// Mitsubishi GX Works2 project: 램프4   PLC: Q02/Q02H

PROGRAM MAIN
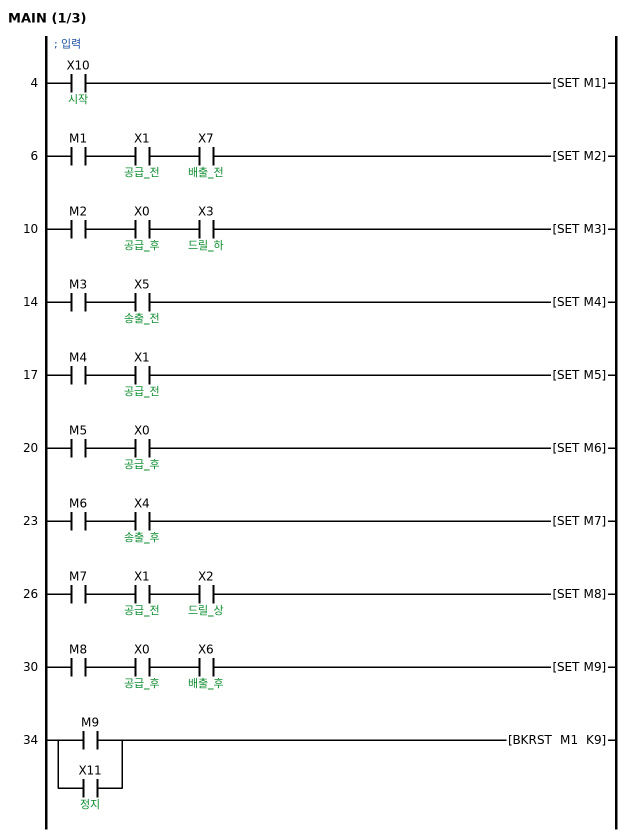
; 입력
4     LD      X10  ; 시작
      SET     M1
6     LD      M1
      AND     X1  ; 공급_전
      AND     X7  ; 배출_전
      SET     M2
10    LD      M2
      AND     X0  ; 공급_후
      AND     X3  ; 드릴_하
      SET     M3
14    LD      M3
      AND     X5  ; 송출_전
      SET     M4
17    LD      M4
      AND     X1  ; 공급_전
      SET     M5
20    LD      M5
      AND     X0  ; 공급_후
      SET     M6
23    LD      M6
      AND     X4  ; 송출_후
      SET     M7
26    LD      M7
      AND     X1  ; 공급_전
      AND     X2  ; 드릴_상
      SET     M8
30    LD      M8
      AND     X0  ; 공급_후
      AND     X6  ; 배출_후
      SET     M9
34    LD      M9
      OR      X11  ; 정지
      BKRST   M1 K9
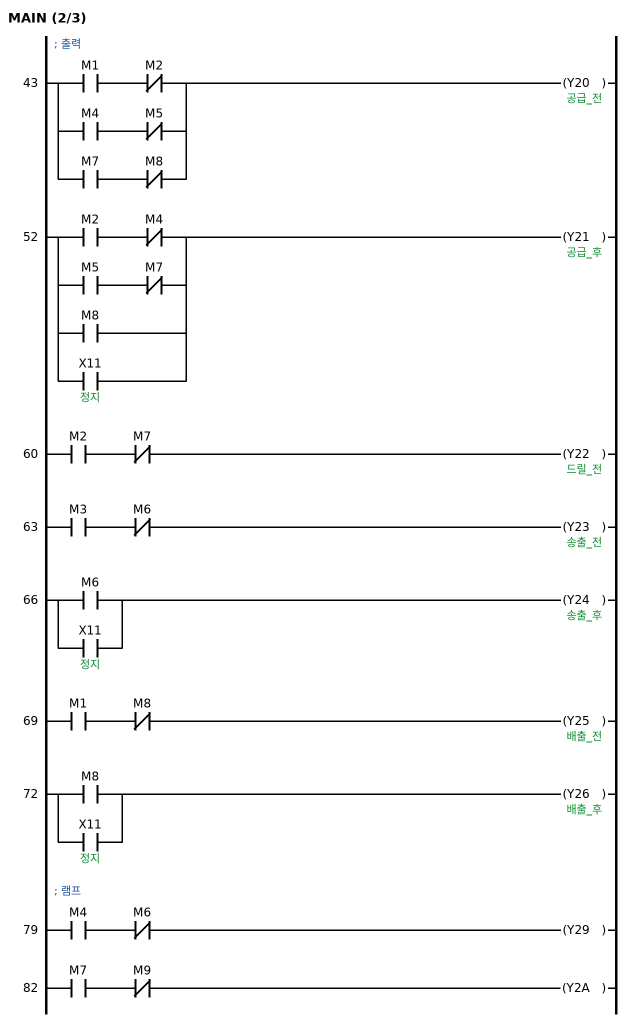
; 출력
43    LD      M1
      ANI     M2
      LD      M4
      ANI     M5
      ORB
      LD      M7
      ANI     M8
      ORB
      OUT     Y20  ; 공급_전
52    LD      M2
      ANI     M4
      LD      M5
      ANI     M7
      ORB
      OR      M8
      OR      X11  ; 정지
      OUT     Y21  ; 공급_후
60    LD      M2
      ANI     M7
      OUT     Y22  ; 드릴_전
63    LD      M3
      ANI     M6
      OUT     Y23  ; 송출_전
66    LD      M6
      OR      X11  ; 정지
      OUT     Y24  ; 송출_후
69    LD      M1
      ANI     M8
      OUT     Y25  ; 배출_전
72    LD      M8
      OR      X11  ; 정지
      OUT     Y26  ; 배출_후
; 램프
79    LD      M4
      ANI     M6
      OUT     Y29
82    LD      M7
      ANI     M9
      OUT     Y2A
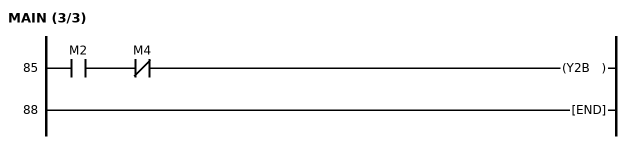
85    LD      M2
      ANI     M4
      OUT     Y2B
88    END
END_PROGRAM
